PROGRAM PRG_LVCP1_Group5
VAR
    // Function Block Instance
    fbContactor: FB_ContactorControl;

    // Contactor 1 IO Structure  
    stContactor_IO: ST_ContactorIO;
    
    // Başlangıç konfigürasyonu için flag
    bContactorInitDone: BOOL := FALSE;
    bCapacitorInitDone: BOOL := FALSE;	
END_VAR



	M_Contactor();
	
	M_Capacitor();

METHOD M_Capacitor : BOOL
VAR
    nGroupIndex : INT;
END_VAR

nGroupIndex := 4;  // Grup 5 için index

IF NOT bCapacitorInitDone THEN
    // Grup 5 değerlerini ata
    GVL_LVCP1.astCompensationGroups[nGroupIndex].rPower := 25.0;
    GVL_LVCP1.astCompensationGroups[nGroupIndex].rVoltage := 450.0;
    GVL_LVCP1.astCompensationGroups[nGroupIndex].nQuantity := 4;
    GVL_LVCP1.astCompensationGroups[nGroupIndex].sTagPrefix := '+EP6-28C1';
    GVL_LVCP1.astCompensationGroups[nGroupIndex].sProductCode := 'ENT.CXD-450-25';
    
    bCapacitorInitDone := TRUE;
END_IF

// Grup 5 aktif durumu
GVL_LVCP1.abGroupActive[nGroupIndex] := stContactor_IO.bFeedback;

M_Capacitor := TRUE;
END_METHOD

METHOD M_Contactor : BOOL
VAR_INPUT
END_VAR
IF NOT bContactorInitDone THEN
    // Konfigürasyon parametreleri
    GVL_LVCP1.stGroup5_ContactorHMI.stConfig.sProjectCode := '+EP6-29K1';
    GVL_LVCP1.stGroup5_ContactorHMI.stConfig.sProductCode := 'SCH LC1G265LSEA';
    GVL_LVCP1.stGroup5_ContactorHMI.stConfig.rRatedCurrent := 265.0;
    GVL_LVCP1.stGroup5_ContactorHMI.stConfig.rRatedVoltage := 1000.0;
    GVL_LVCP1.stGroup5_ContactorHMI.stConfig.nPhaseCount := 3;
    GVL_LVCP1.stGroup5_ContactorHMI.stConfig.tFeedbackDelay := T#500MS;
    GVL_LVCP1.stGroup5_ContactorHMI.stConfig.tWeldedDelay := T#2S;
    GVL_LVCP1.stGroup5_ContactorHMI.stConfig.dwOperationLimit := 100000;
    
    // Başlangıç bakım sayacı
    GVL_LVCP1.stGroup5_ContactorHMI.stStatistics.dwRemainingOperations := GVL_LVCP1.stGroup5_ContactorHMI.stConfig.dwOperationLimit;
    
    bContactorInitDone := TRUE;
END_IF

// Function Block Çağrısı
fbContactor(
    // Fiziksel Girişler
    bFeedback := stContactor_IO.bFeedback,
    bPLCControl := stContactor_IO.bPLCControl,
    
    // Güvenlik Girişleri
    bSafetyLoop := GVL_Alarm.bSafetyLoop,
    bInterlock := FALSE,
    
    // Sistem Girişleri
    bMasterReset := GVL_Alarm.bMasterReset,
    
    // HMI Bağlantısı
    stHMI := GVL_LVCP1.stGroup5_ContactorHMI,
    
    // Fiziksel Çıkış
    bOutput => stContactor_IO.bOutput
);

M_Contactor := TRUE;
END_METHOD

END_PROGRAM

(* stored: Version 1.1.0.1, ProductVersion 3.1.4024.15
   POU PRG_LVCP1_Group5: Id {97b39ed4-3af7-4775-bb97-b13d10a0ef01}, SpecialFunc None
   Method M_Capacitor: Id {5baaf4db-781e-45ae-879c-80c4f22982da}
   Method M_Contactor: Id {f3e77aed-46bd-49e0-9efc-5368b8bb2e81} *)
